FUNCTION ErrorStep : UDINT
VAR_IN_OUT
	StateVar : UDINT;
END_VAR

ErrorStep := StateVar := ((StateVar / 10) * 10) + 9;

END_FUNCTION

(* stored: Version 1.1.0.1, ProductVersion 3.1.4024.13
   POU ErrorStep: Id {858799b2-f3f9-45e8-ae72-f37c535cc7a6}, SpecialFunc None *)
